Yaskawa INFORM job: UNTITLED.JBI

/JOB
//NAME UNTITLED
///FOLDERNAME INNE
//POS
///NPOS 0,0,0,0,0,0
//INST
///DATE 2023/10/04 15:12
///ATTR SC,RW
///GROUP1 RB1,BS1
NOP
'UNTITLED
CALL JOB:R2_W8
CALL JOB:R2_W11
CALL JOB:R2_W13
CALL JOB:R2_W2
CALL JOB:R2_W4
CALL JOB:R2_W6
END
